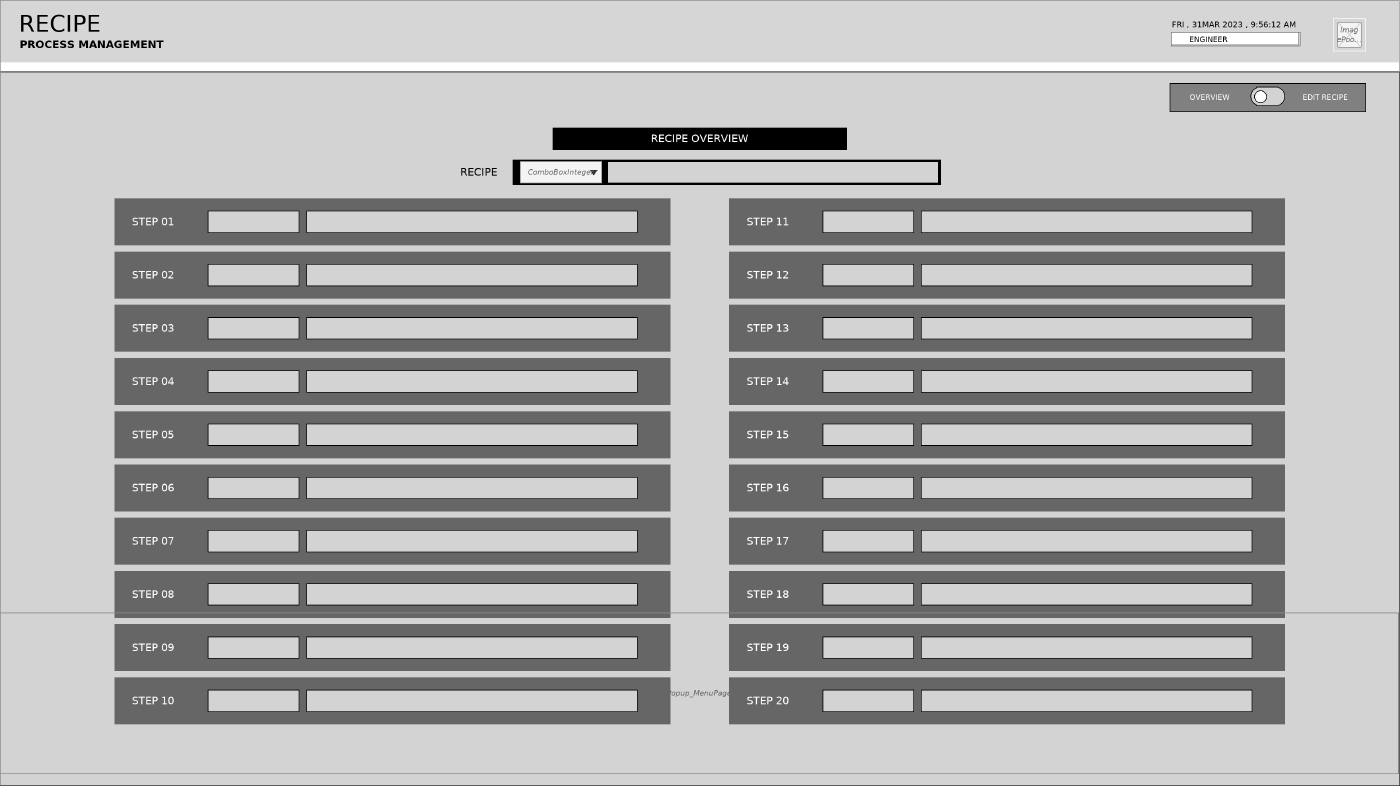
VISUALIZATION Recipe_Page  // 1920x1078
    Rectangle (0,98 1920x980)
    Rectangle (0,63 1920x26)
        p3528305787: HMI_Ctrl.ANIMATION3
    Rectangle (0,0 1919x85)
    Label (23,6 267x53), "RECIPE"
    Label (24,49 320x24), "PROCESS MANAGEMENT"
    Group (1604,25 188x38)
        Label (0,0 188x18), "FRI , 31MAR 2023 , 9:56:12 AM"
        Button (2,19 177x19), image: VisuSymbols.Symbols.AddUser
        Label (24,23 91x12), "ENGINEER"
    RoundedRectangle (157,272 762x64)
    Label (178,292 103x24), "STEP 01"
    RoundedRectangle (285,289 125x30)
    RoundedRectangle (420,289 454x30)
    RoundedRectangle (157,345 762x64)
    Label (178,365 103x24), "STEP 02"
    RoundedRectangle (285,362 125x30)
    RoundedRectangle (420,362 454x30)
    RoundedRectangle (157,418 762x64)
    Label (178,438 103x24), "STEP 03"
    RoundedRectangle (285,435 125x30)
    RoundedRectangle (420,435 454x30)
    RoundedRectangle (157,491 762x64)
    Label (178,511 103x24), "STEP 04"
    RoundedRectangle (285,508 125x30)
    RoundedRectangle (420,508 454x30)
    RoundedRectangle (157,564 762x64)
    Label (178,584 103x24), "STEP 05"
    RoundedRectangle (285,581 125x30)
    RoundedRectangle (420,581 454x30)
    RoundedRectangle (157,637 762x64)
    Label (178,657 103x24), "STEP 06"
    RoundedRectangle (285,654 125x30)
    RoundedRectangle (420,654 454x30)
    RoundedRectangle (157,710 762x64)
    Label (178,730 103x24), "STEP 07"
    RoundedRectangle (285,727 125x30)
    RoundedRectangle (420,727 454x30)
    RoundedRectangle (157,783 762x64)
    Label (178,803 103x24), "STEP 08"
    RoundedRectangle (285,800 125x30)
    RoundedRectangle (420,800 454x30)
    RoundedRectangle (157,856 762x64)
    Label (178,876 103x24), "STEP 09"
    RoundedRectangle (285,873 125x30)
    RoundedRectangle (420,873 454x30)
    RoundedRectangle (157,929 762x64)
    Label (178,949 103x24), "STEP 10"
    RoundedRectangle (285,946 125x30)
    RoundedRectangle (420,946 454x30)
    RoundedRectangle (1000,272 762x64)
    Label (1021,292 103x24), "STEP 11"
    RoundedRectangle (1128,289 125x30)
    RoundedRectangle (1263,289 454x30)
    RoundedRectangle (1000,345 762x64)
    Label (1021,365 103x24), "STEP 12"
    RoundedRectangle (1128,362 125x30)
    RoundedRectangle (1263,362 454x30)
    RoundedRectangle (1000,418 762x64)
    Label (1021,438 103x24), "STEP 13"
    RoundedRectangle (1128,435 125x30)
    RoundedRectangle (1263,435 454x30)
    RoundedRectangle (1000,491 762x64)
    Label (1021,511 103x24), "STEP 14"
    RoundedRectangle (1128,508 125x30)
    RoundedRectangle (1263,508 454x30)
    RoundedRectangle (1000,564 762x64)
    Label (1021,584 103x24), "STEP 15"
    RoundedRectangle (1128,581 125x30)
    RoundedRectangle (1263,581 454x30)
    RoundedRectangle (1000,637 762x64)
    Label (1021,657 103x24), "STEP 16"
    RoundedRectangle (1128,654 125x30)
    RoundedRectangle (1263,654 454x30)
    RoundedRectangle (1000,710 762x64)
    Label (1021,730 103x24), "STEP 17"
    RoundedRectangle (1128,727 125x30)
    RoundedRectangle (1263,727 454x30)
    RoundedRectangle (1000,783 762x64)
    Label (1021,803 103x24), "STEP 18"
    RoundedRectangle (1128,800 125x30)
    RoundedRectangle (1263,800 454x30)
    RoundedRectangle (1000,856 762x64)
    Label (1021,876 103x24), "STEP 19"
    RoundedRectangle (1128,873 125x30)
    RoundedRectangle (1263,873 454x30)
    RoundedRectangle (1000,929 762x64)
    Label (1021,949 103x24), "STEP 20"
    RoundedRectangle (1128,946 125x30)
    RoundedRectangle (1263,946 454x30)
    Rectangle (758,175 403x30), "RECIPE OVERVIEW"
    RoundedRectangle (703,219 587x34)
    RoundedRectangle (833,221 454x30)
    ComboBoxInteger (713,221 112x30)
    Label (628,224 103x24), "RECIPE"
    Group (1828,25 45x45)
        OnMouseClick: toggle HMI_Ctrl.MenuButton
        RoundedRectangle (0,0 45x45), colour toggle: HMI_Ctrl.MenuButton
        Image (6,5 33x35), image: ImagePool.Menu Button
    Group (1604,113 269x41)
        RoundedRectangle (0,1 269x39)
        Label (1,0 108x41), "OVERVIEW"
        Label (161,0 105x41), "EDIT RECIPE"
        Group (111,6 47x26)
            OnMouseClick: change screen: RecipeSSUR_Page
            Group (0,0 47x26)
                Ellipse (0,0 26x26)
                Ellipse (21,0 26x26)
                RoundedRectangle (8,0 29x26)
            Ellipse (1,1 24x24)
            Ellipse (23,1 23x24)
            RoundedRectangle (9,1 28x24)
            Ellipse (5,5 17x17)
    Frame (0,840 1918x221), invisible if: HMI_Ctrl.CloseMenuButton
        shows Popup_MenuPage()
END_VISUALIZATION

(* stored: Version 1.1.0.1, ProductVersion 3.1.4024.12
   Visu Recipe_Page: Id {6834e29c-8f5b-4c3a-b3b7-1399abe23f71} *)
